// TIA Portal V16 export
// export: Created 2021-11-12T13:31:46.8533956Z, ExportSetting WithDefaults, DisplayName Totally Integrated Automation Portal, DisplayVersion V16 Update 3, DisplayName TIA Portal Version Control Interface, DisplayVersion V16 Update 2, DisplayName TIA Portal Openness, DisplayVersion V16 Update 3, DisplayName SINAMICS Startdrive Advanced, DisplayVersion V16 Update 5, DisplayName SINAMICS Startdrive G130, G150, S120, S150, SINAMICS MV, S210, DisplayVersion V16 Update 5, DisplayName SINAMICS Startdrive G110M, G120, G120C, G120D, G120P, G115D, DisplayVersion V16 Update 5, DisplayName STEP 7 Professional, DisplayVersion V16 Update 3, DisplayName STEP 7 Safety, DisplayVersion V16, DisplayName WinCC UA Professional, DisplayVersion V16 Update 3
FUNCTION "Inputs" : Void   // FC3, LAD
TITLE = FC Inputs
{ S7_Optimized_Access := 'TRUE' }
VERSION : 0.1
// MICE Wood tempate block
// Call FBs that reads data from Input modules
// every single FB for 1 decentral device like ET200
// No logic in this block
// stored: AutoNumber false, IsIECCheckEnabled false, SetENOAutomatically false, UDAEnableTagReadback false
BEGIN

REGION Network 1: IM_000+UH01-KF10
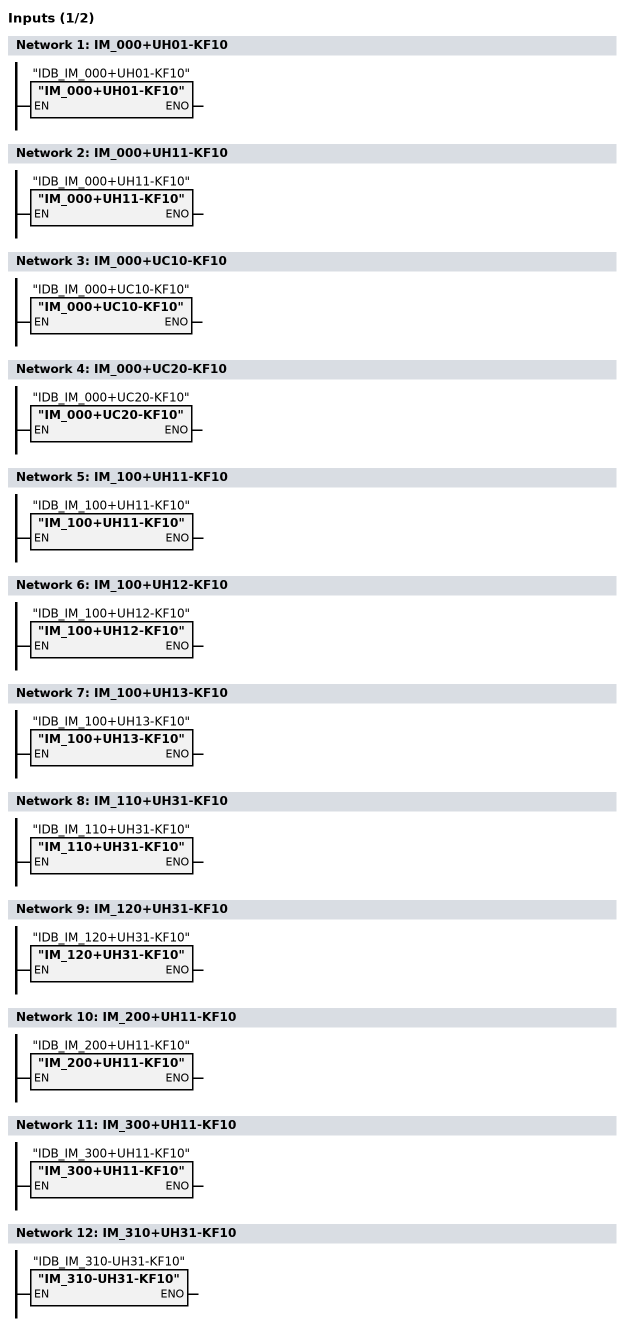
   RUNG wire#powerrail
      "IDB_IM_000+UH01-KF10"()
   END_RUNG
   // the same network as SCL:
   "IDB_IM_000+UH01-KF10"();   // "IM_000+UH01-KF10"
END_REGION

REGION Network 2: IM_000+UH11-KF10
   RUNG wire#powerrail
      "IDB_IM_000+UH11-KF10"()
   END_RUNG
   // the same network as SCL:
   "IDB_IM_000+UH11-KF10"();   // "IM_000+UH11-KF10"
END_REGION

REGION Network 3: IM_000+UC10-KF10
   RUNG wire#powerrail
      "IDB_IM_000+UC10-KF10"()
   END_RUNG
   // the same network as SCL:
   "IDB_IM_000+UC10-KF10"();   // "IM_000+UC10-KF10"
END_REGION

REGION Network 4: IM_000+UC20-KF10
   RUNG wire#powerrail
      "IDB_IM_000+UC20-KF10"()
   END_RUNG
   // the same network as SCL:
   "IDB_IM_000+UC20-KF10"();   // "IM_000+UC20-KF10"
END_REGION

REGION Network 5: IM_100+UH11-KF10
   RUNG wire#powerrail
      "IDB_IM_100+UH11-KF10"()
   END_RUNG
   // the same network as SCL:
   "IDB_IM_100+UH11-KF10"();   // "IM_100+UH11-KF10"
END_REGION

REGION Network 6: IM_100+UH12-KF10
   RUNG wire#powerrail
      "IDB_IM_100+UH12-KF10"()
   END_RUNG
   // the same network as SCL:
   "IDB_IM_100+UH12-KF10"();   // "IM_100+UH12-KF10"
END_REGION

REGION Network 7: IM_100+UH13-KF10
   RUNG wire#powerrail
      "IDB_IM_100+UH13-KF10"()
   END_RUNG
   // the same network as SCL:
   "IDB_IM_100+UH13-KF10"();   // "IM_100+UH13-KF10"
END_REGION

REGION Network 8: IM_110+UH31-KF10
   RUNG wire#powerrail
      "IDB_IM_110+UH31-KF10"()
   END_RUNG
   // the same network as SCL:
   "IDB_IM_110+UH31-KF10"();   // "IM_110+UH31-KF10"
END_REGION

REGION Network 9: IM_120+UH31-KF10
   RUNG wire#powerrail
      "IDB_IM_120+UH31-KF10"()
   END_RUNG
   // the same network as SCL:
   "IDB_IM_120+UH31-KF10"();   // "IM_120+UH31-KF10"
END_REGION

REGION Network 10: IM_200+UH11-KF10
   RUNG wire#powerrail
      "IDB_IM_200+UH11-KF10"()
   END_RUNG
   // the same network as SCL:
   "IDB_IM_200+UH11-KF10"();   // "IM_200+UH11-KF10"
END_REGION

REGION Network 11: IM_300+UH11-KF10
   RUNG wire#powerrail
      "IDB_IM_300+UH11-KF10"()
   END_RUNG
   // the same network as SCL:
   "IDB_IM_300+UH11-KF10"();   // "IM_300+UH11-KF10"
END_REGION

REGION Network 12: IM_310+UH31-KF10
   RUNG wire#powerrail
      "IDB_IM_310-UH31-KF10"()
   END_RUNG
   // the same network as SCL:
   "IDB_IM_310-UH31-KF10"();   // "IM_310-UH31-KF10"
END_REGION

REGION Network 13: IM_400+UH11-KF10
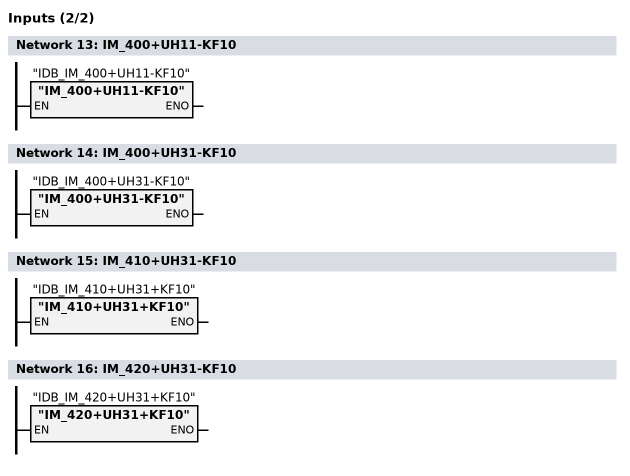
   RUNG wire#powerrail
      "IDB_IM_400+UH11-KF10"()
   END_RUNG
   // the same network as SCL:
   "IDB_IM_400+UH11-KF10"();   // "IM_400+UH11-KF10"
END_REGION

REGION Network 14: IM_400+UH31-KF10
   RUNG wire#powerrail
      "IDB_IM_400+UH31-KF10"()
   END_RUNG
   // the same network as SCL:
   "IDB_IM_400+UH31-KF10"();   // "IM_400+UH31-KF10"
END_REGION

REGION Network 15: IM_410+UH31-KF10
   RUNG wire#powerrail
      "IDB_IM_410+UH31+KF10"()
   END_RUNG
   // the same network as SCL:
   "IDB_IM_410+UH31+KF10"();   // "IM_410+UH31+KF10"
END_REGION

REGION Network 16: IM_420+UH31-KF10
   RUNG wire#powerrail
      "IDB_IM_420+UH31+KF10"()
   END_RUNG
   // the same network as SCL:
   "IDB_IM_420+UH31+KF10"();   // "IM_420+UH31+KF10"
END_REGION
END_FUNCTION
